PROGRAM Axe_06_A	//Rotation angulaire laser
VAR
	ALaser	:FB_Axe_A_Ethercat_V1_1;
	test1: BOOL;
END_VAR

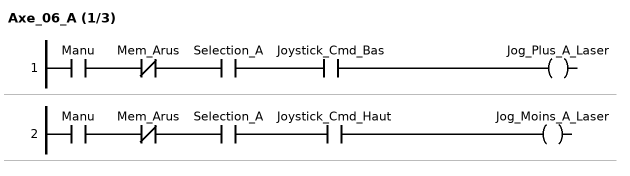
// NETWORK 1
Jog_Plus_A_Laser := Manu AND NOT Mem_Arus AND Selection_A AND Joystick_Cmd_Bas;

// NETWORK 2
Jog_Moins_A_Laser := Manu AND NOT Mem_Arus AND Selection_A AND Joystick_Cmd_Haut;

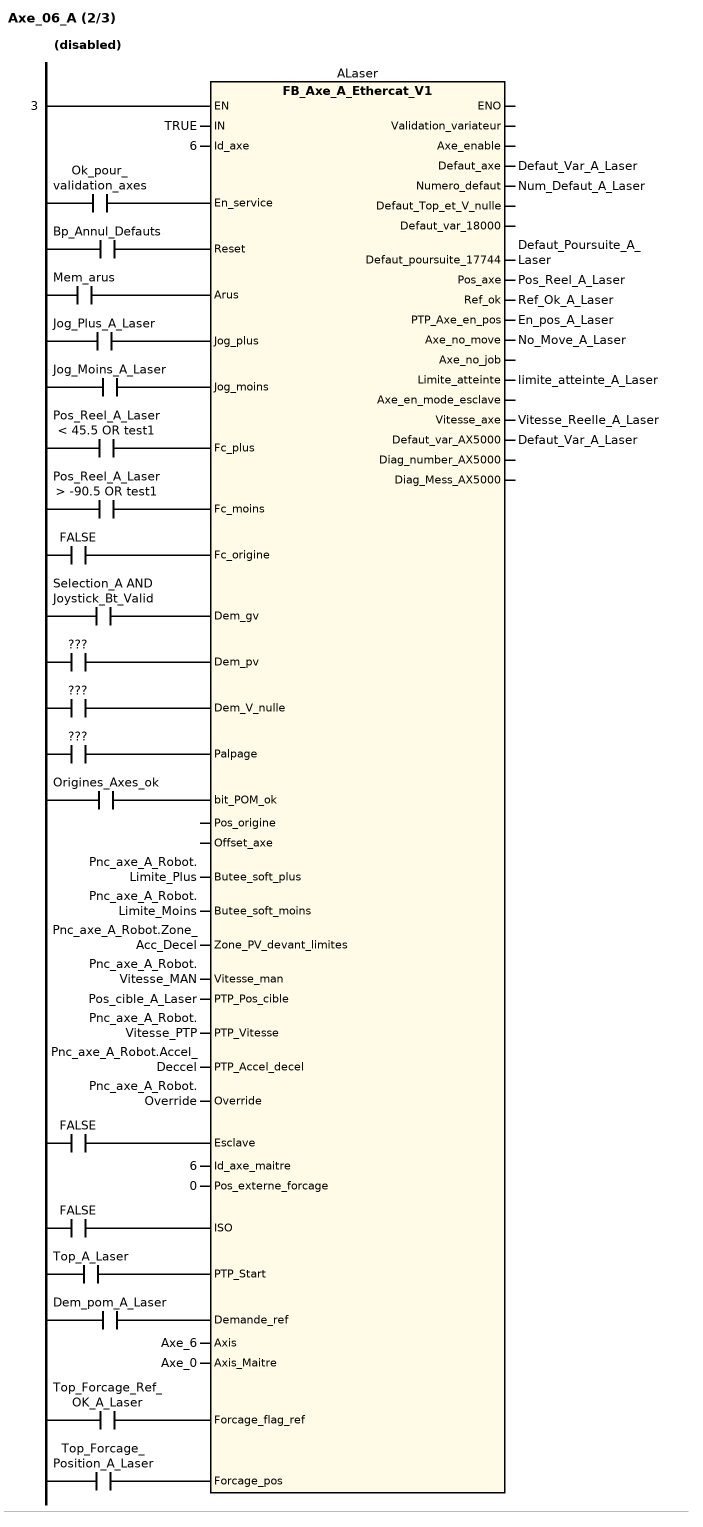
// NETWORK 3 (disabled)
// ALaser(
//     IN := TRUE,
//     Id_axe := 6,
//     En_service := Ok_pour_validation_axes,
//     Reset := Bp_Annul_Defauts,
//     Arus := Mem_arus,
//     Jog_plus := Jog_Plus_A_Laser,
//     Jog_moins := Jog_Moins_A_Laser,
//     Fc_plus := Pos_Reel_A_Laser < 45.5 OR test1,
//     Fc_moins := Pos_Reel_A_Laser > -90.5 OR test1,
//     Fc_origine := FALSE,
//     Dem_gv := Selection_A AND Joystick_Bt_Valid,
//     bit_POM_ok := Origines_Axes_ok,
//     Butee_soft_plus := Pnc_axe_A_Robot.Limite_Plus,
//     Butee_soft_moins := Pnc_axe_A_Robot.Limite_Moins,
//     Zone_PV_devant_limites := Pnc_axe_A_Robot.Zone_Acc_Decel,
//     Vitesse_man := Pnc_axe_A_Robot.Vitesse_MAN,
//     PTP_Pos_cible := Pos_cible_A_Laser,
//     PTP_Vitesse := Pnc_axe_A_Robot.Vitesse_PTP,
//     PTP_Accel_decel := Pnc_axe_A_Robot.Accel_Deccel,
//     Override := Pnc_axe_A_Robot.Override,
//     Esclave := FALSE,
//     Id_axe_maitre := 6,
//     Pos_externe_forcage := 0,
//     ISO := FALSE,
//     PTP_Start := Top_A_Laser,
//     Demande_ref := Dem_pom_A_Laser,
//     Axis := Axe_6,
//     Axis_Maitre := Axe_0,
//     Forcage_flag_ref := Top_Forcage_Ref_OK_A_Laser,
//     Forcage_pos := Top_Forcage_Position_A_Laser,
//     Defaut_axe => Defaut_Var_A_Laser,
//     Numero_defaut => Num_Defaut_A_Laser,
//     Defaut_poursuite_17744 => Defaut_Poursuite_A_Laser,
//     Pos_axe => Pos_Reel_A_Laser,
//     Ref_ok => Ref_Ok_A_Laser,
//     PTP_Axe_en_pos => En_pos_A_Laser,
//     Axe_no_move => No_Move_A_Laser,
//     Limite_atteinte => limite_atteinte_A_Laser,
//     Vitesse_axe => Vitesse_Reelle_A_Laser,
//     Defaut_var_AX5000 => Defaut_Var_A_Laser); // FB_Axe_A_Ethercat_V1

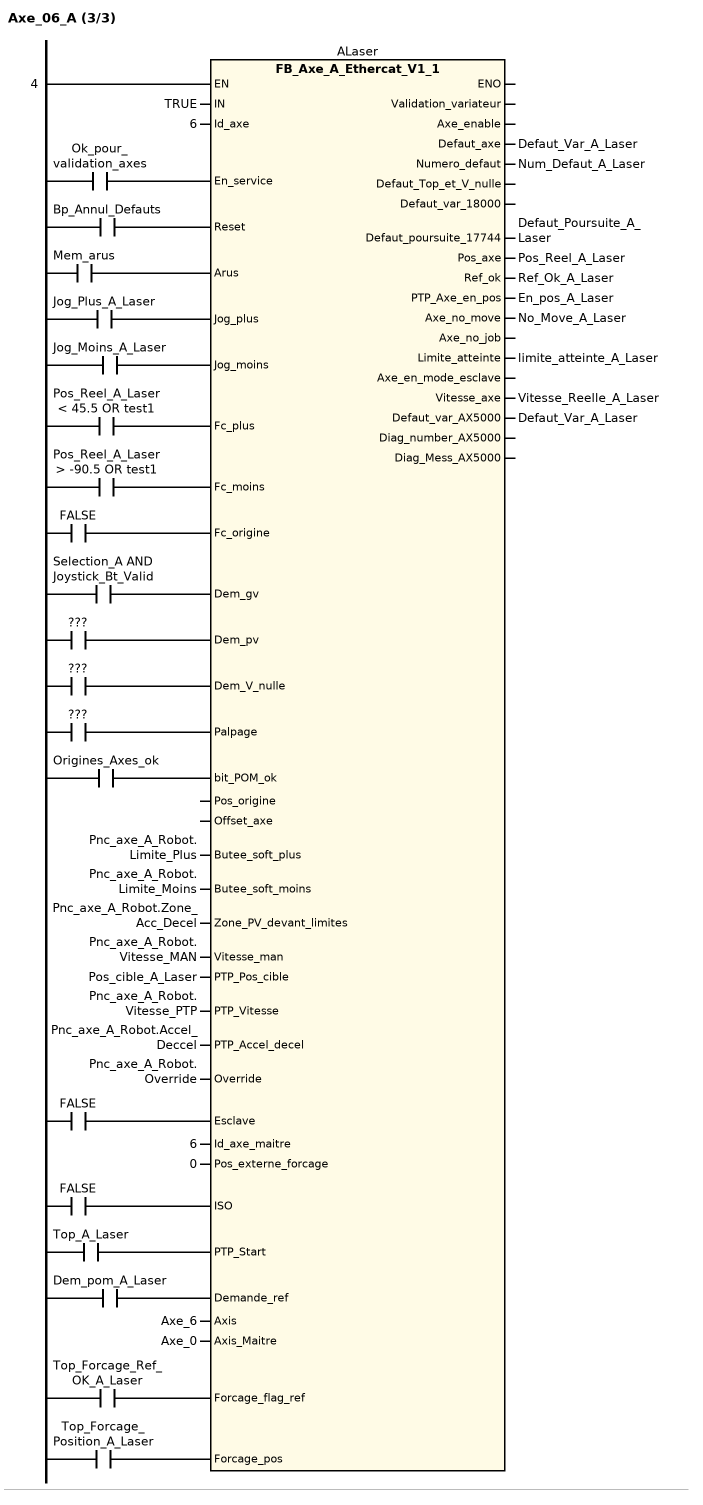
// NETWORK 4
ALaser(
    IN := TRUE,
    Id_axe := 6,
    En_service := Ok_pour_validation_axes,
    Reset := Bp_Annul_Defauts,
    Arus := Mem_arus,
    Jog_plus := Jog_Plus_A_Laser,
    Jog_moins := Jog_Moins_A_Laser,
    Fc_plus := Pos_Reel_A_Laser < 45.5 OR test1,
    Fc_moins := Pos_Reel_A_Laser > -90.5 OR test1,
    Fc_origine := FALSE,
    Dem_gv := Selection_A AND Joystick_Bt_Valid,
    bit_POM_ok := Origines_Axes_ok,
    Butee_soft_plus := Pnc_axe_A_Robot.Limite_Plus,
    Butee_soft_moins := Pnc_axe_A_Robot.Limite_Moins,
    Zone_PV_devant_limites := Pnc_axe_A_Robot.Zone_Acc_Decel,
    Vitesse_man := Pnc_axe_A_Robot.Vitesse_MAN,
    PTP_Pos_cible := Pos_cible_A_Laser,
    PTP_Vitesse := Pnc_axe_A_Robot.Vitesse_PTP,
    PTP_Accel_decel := Pnc_axe_A_Robot.Accel_Deccel,
    Override := Pnc_axe_A_Robot.Override,
    Esclave := FALSE,
    Id_axe_maitre := 6,
    Pos_externe_forcage := 0,
    ISO := FALSE,
    PTP_Start := Top_A_Laser,
    Demande_ref := Dem_pom_A_Laser,
    Axis := Axe_6,
    Axis_Maitre := Axe_0,
    Forcage_flag_ref := Top_Forcage_Ref_OK_A_Laser,
    Forcage_pos := Top_Forcage_Position_A_Laser,
    Defaut_axe => Defaut_Var_A_Laser,
    Numero_defaut => Num_Defaut_A_Laser,
    Defaut_poursuite_17744 => Defaut_Poursuite_A_Laser,
    Pos_axe => Pos_Reel_A_Laser,
    Ref_ok => Ref_Ok_A_Laser,
    PTP_Axe_en_pos => En_pos_A_Laser,
    Axe_no_move => No_Move_A_Laser,
    Limite_atteinte => limite_atteinte_A_Laser,
    Vitesse_axe => Vitesse_Reelle_A_Laser,
    Defaut_var_AX5000 => Defaut_Var_A_Laser); // FB_Axe_A_Ethercat_V1_1

END_PROGRAM

(* stored: Version 1.1.0.1
   POU Axe_06_A: Id {a446512a-96b4-4e5c-99bc-e9ea8dad01a1}, SpecialFunc None *)
